(* IEC 61131-3 sources: vertical-injection-machine-docs/docs/IM_SYS_PRG/Code/Modbus通讯, 2 files *)

(* ---- ModbusTypes.st ---- *)
(*
  ModbusTypes.st
  功能：
  1. 定义整机唯一的 Modbus 通讯镜像边界，统一收口 HMI 参数区与面板按键/灯区。
  2. 让 PLC 内部业务边界与外部 Modbus 通讯边界彻底解耦，后续只在本层处理寄存器地址和协议兼容。
  3. 为 `FB_Modbus` 提供统一的数据结构，避免 HMI 与面板继续维护两套分散的通讯类型。

  说明：
  1. `ST_Modbus` 是当前工程唯一允许直接绑定真实 Modbus 寄存器区的公共边界。
  2. `ST_HMIProcessPara`、`ST_HMIParaCommand`、`ST_HMIParaStatus`、`ST_PanelIO` 仍然只表示 PLC 内部业务边界。
  3. 后续若需要调整寄存器地址、拆装报文或兼容多个 HMI/面板协议版本，应优先扩展本文件与 `FB_Modbus`，不要回流到业务块。
*)

TYPE ST_ModbusHMIInput :
STRUCT
    stPara: ST_HMIProcessPara;        // HMI 通过 Modbus 写给 PLC 的参数编辑区镜像；由 `FB_Modbus` 在输入绑定阶段写入 PLC 内部 HMI 参数业务边界。
    stCommand: ST_HMIParaCommand;     // HMI 通过 Modbus 写给 PLC 的参数命令区镜像；由 `FB_Modbus` 在输入绑定阶段写入 PLC 内部 HMI 命令边界。
END_STRUCT
END_TYPE

TYPE ST_ModbusHMIOutput :
STRUCT
    stPara: ST_HMIProcessPara;        // PLC 通过 Modbus 回写给 HMI 的参数镜像区；供画面读取当前 PLC 认可的参数缓冲区。
    stStatus: ST_HMIParaStatus;       // PLC 通过 Modbus 回写给 HMI 的参数状态区；供画面读取参数同步结果、拦截原因与脏标记。
END_STRUCT
END_TYPE

TYPE ST_ModbusPanelInput :
STRUCT
    uiIN0: UINT;                      // 面板/HMI 通过 Modbus 写给 PLC 的输入字 0；承载排序号 `1..16` 对应的 16 个按键位。
    uiIN1: UINT;                      // 面板/HMI 通过 Modbus 写给 PLC 的输入字 1；承载排序号 `17..32` 对应的 16 个按键位。
    uiIN2: UINT;                      // 面板/HMI 通过 Modbus 写给 PLC 的输入字 2；承载排序号 `33..48` 对应的 16 个按键位。
    uiIN3: UINT;                      // 面板/HMI 通过 Modbus 写给 PLC 的输入字 3；承载排序号 `49..64` 对应的 16 个按键位。
END_STRUCT
END_TYPE

TYPE ST_ModbusPanelOutput :
STRUCT
    uiOUT0: UINT;                     // PLC 通过 Modbus 回写给面板/HMI 的输出字 0；承载排序号 `1..16` 对应的 16 个灯位。
    uiOUT1: UINT;                     // PLC 通过 Modbus 回写给面板/HMI 的输出字 1；承载排序号 `17..32` 对应的 16 个灯位。
    uiOUT2: UINT;                     // PLC 通过 Modbus 回写给面板/HMI 的输出字 2；承载排序号 `33..48` 对应的 16 个灯位。
    uiOUT3: UINT;                     // PLC 通过 Modbus 回写给面板/HMI 的输出字 3；承载排序号 `49..64` 对应的 16 个灯位。
END_STRUCT
END_TYPE

TYPE ST_Modbus :
STRUCT
    stHMIInput: ST_ModbusHMIInput;    // HMI -> PLC 的统一 Modbus 输入镜像区；收口参数编辑区与参数命令区。
    stHMIOutput: ST_ModbusHMIOutput;  // PLC -> HMI 的统一 Modbus 输出镜像区；收口参数缓冲区与参数状态区。
    stPanelInput: ST_ModbusPanelInput; // 面板/HMI -> PLC 的统一 Modbus 输入镜像区；收口 4 个原始按键输入字。
    stPanelOutput: ST_ModbusPanelOutput; // PLC -> 面板/HMI 的统一 Modbus 输出镜像区；收口 4 个原始灯输出字。
END_STRUCT
END_TYPE

(* ---- FB_Modbus.st ---- *)
(*
  FB_Modbus 功能块
  功能：
  1. 统一处理整机 Modbus 通讯镜像与 PLC 内部业务边界之间的双向绑定。
  2. 输入阶段负责把 HMI 参数区和面板按键字从 `ST_Modbus` 写入 PLC 内部边界。
  3. 输出阶段负责把 PLC 内部 HMI 状态和面板灯字回写到 `ST_Modbus`。

  调用要求：
  1. 应由 `PRG_MainControl` 在每个扫描周期至少调用两次：业务块前执行输入绑定，业务块后执行输出绑定。
  2. `bBindInput` 与 `bBindOutput` 可独立控制；若同拍同时为 TRUE，则本块会先做输入绑定，再做输出绑定。
  3. 真实 Modbus 驱动、寄存器地址表和协议版本兼容层只允许绑定在 `stModbus` 上，不允许散写到其他业务块。
*)
FUNCTION_BLOCK FB_Modbus
VAR_INPUT
    bBindInput: BOOL;                 // TRUE=本次调用执行“Modbus 通讯镜像 -> PLC 内部业务边界”的输入绑定阶段。
    bBindOutput: BOOL;                // TRUE=本次调用执行“PLC 内部业务边界 -> Modbus 通讯镜像”的输出绑定阶段。
END_VAR
VAR_IN_OUT
    stModbus: ST_Modbus;              // 顶层唯一统一 Modbus 通讯镜像边界；实际通讯驱动应直接绑定到这个结构。
    stHMIPara: ST_HMIProcessPara;     // PLC 内部 HMI 参数业务边界；输入绑定阶段回写，输出绑定阶段回读。
    stHMICommand: ST_HMIParaCommand;  // PLC 内部 HMI 参数命令业务边界；输入绑定阶段回写，供 HMI 参数接口块消费。
    stHMIStatus: ST_HMIParaStatus;    // PLC 内部 HMI 参数状态业务边界；输出绑定阶段回读，供 HMI 画面显示。
    stPanelIO: ST_PanelIO;            // PLC 内部面板原始字边界；输入绑定阶段回写按键字，输出绑定阶段回读灯字。
END_VAR

IF bBindInput THEN
    stHMIPara := stModbus.stHMIInput.stPara;            // 把统一 Modbus HMI 输入区中的参数编辑镜像拷贝到 PLC 内部 HMI 参数业务边界。
    stHMICommand := stModbus.stHMIInput.stCommand;      // 把统一 Modbus HMI 输入区中的参数命令镜像拷贝到 PLC 内部 HMI 命令业务边界。
    stPanelIO.uiIN0 := stModbus.stPanelInput.uiIN0;     // 把统一 Modbus 面板输入区中的输入字 0 拷贝到 PLC 内部面板输入字 0。
    stPanelIO.uiIN1 := stModbus.stPanelInput.uiIN1;     // 把统一 Modbus 面板输入区中的输入字 1 拷贝到 PLC 内部面板输入字 1。
    stPanelIO.uiIN2 := stModbus.stPanelInput.uiIN2;     // 把统一 Modbus 面板输入区中的输入字 2 拷贝到 PLC 内部面板输入字 2。
    stPanelIO.uiIN3 := stModbus.stPanelInput.uiIN3;     // 把统一 Modbus 面板输入区中的输入字 3 拷贝到 PLC 内部面板输入字 3。
END_IF;

IF bBindOutput THEN
    stModbus.stHMIOutput.stPara := stHMIPara;           // 把 PLC 当前认可的 HMI 参数缓冲区镜像回写到统一 Modbus HMI 输出区。
    stModbus.stHMIOutput.stStatus := stHMIStatus;       // 把 PLC 当前 HMI 参数状态镜像回写到统一 Modbus HMI 输出区。
    stModbus.stPanelOutput.uiOUT0 := stPanelIO.uiOUT0;  // 把 PLC 内部面板灯输出字 0 回写到统一 Modbus 面板输出区。
    stModbus.stPanelOutput.uiOUT1 := stPanelIO.uiOUT1;  // 把 PLC 内部面板灯输出字 1 回写到统一 Modbus 面板输出区。
    stModbus.stPanelOutput.uiOUT2 := stPanelIO.uiOUT2;  // 把 PLC 内部面板灯输出字 2 回写到统一 Modbus 面板输出区。
    stModbus.stPanelOutput.uiOUT3 := stPanelIO.uiOUT3;  // 把 PLC 内部面板灯输出字 3 回写到统一 Modbus 面板输出区。
END_IF;
END_FUNCTION_BLOCK
